ABB RAPID module: backup.MOD

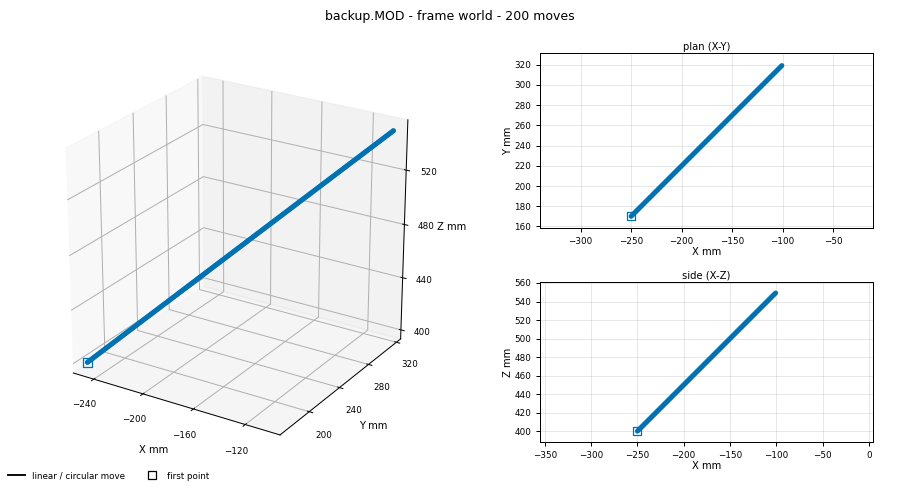
[picture p0: tool path of backup.MOD in frame world, 200 of 201 moves have a stored position in this frame; points joined in program order, loops and branches not executed]
MODULE MainModule
PERS tooldata Servo:=[TRUE,[[0,0,114.2],[1,0,0,0]],[0.215,[8.7,12.3,49.2],[1,0,0,0],0.00021,0.00024,0.00009]];
PERS tooldata tObject:=[TRUE,[[0,0,130],[0.707106781,-0.707106781,0,0]],[0.215,[8.7,12.3,49.2],[1,0,0,0],0.00021,0.00024,0.00009]];
PERS wobjdata handpos:= [FALSE,TRUE,"",[[-400,20,250],[1,0,0,0]],[[0,0,0],[1,0,0,0]]];


    PROC main()
        ConfL\Off;
        SingArea\Wrist;
        !Startpos
        MoveAbsJ [[95.3526,8.2285,12.3495,-7.77934,80.6461,5.41418],[87.0554,9E+09,9E+09,9E+09,9E+09,9E+09]] \NoEOffs, v1000, fine, wi_tGripper;
	    path;
    ENDPROC
    PROC path()

VAR robtarget t0 := [[150.0, 150.0, 150.0], [0, -1, 0, 0], [0,0,-1,4], [-96,9E+09,9E+09,9E+09,9E+09,9E+09]];
VAR robtarget t1 := [[150.75, 150.75, 150.75], [0, -1, 0, 0], [0,0,-1,4], [-96,9E+09,9E+09,9E+09,9E+09,9E+09]];
VAR robtarget t2 := [[151.5, 151.5, 151.5], [0, -1, 0, 0], [0,0,-1,4], [-96,9E+09,9E+09,9E+09,9E+09,9E+09]];
VAR robtarget t3 := [[152.25, 152.25, 152.25], [0, -1, 0, 0], [0,0,-1,4], [-96,9E+09,9E+09,9E+09,9E+09,9E+09]];
VAR robtarget t4 := [[153.0, 153.0, 153.0], [0, -1, 0, 0], [0,0,-1,4], [-96,9E+09,9E+09,9E+09,9E+09,9E+09]];
VAR robtarget t5 := [[153.75, 153.75, 153.75], [0, -1, 0, 0], [0,0,-1,4], [-96,9E+09,9E+09,9E+09,9E+09,9E+09]];
VAR robtarget t6 := [[154.5, 154.5, 154.5], [0, -1, 0, 0], [0,0,-1,4], [-96,9E+09,9E+09,9E+09,9E+09,9E+09]];
VAR robtarget t7 := [[155.25, 155.25, 155.25], [0, -1, 0, 0], [0,0,-1,4], [-96,9E+09,9E+09,9E+09,9E+09,9E+09]];
VAR robtarget t8 := [[156.0, 156.0, 156.0], [0, -1, 0, 0], [0,0,-1,4], [-96,9E+09,9E+09,9E+09,9E+09,9E+09]];
VAR robtarget t9 := [[156.75, 156.75, 156.75], [0, -1, 0, 0], [0,0,-1,4], [-96,9E+09,9E+09,9E+09,9E+09,9E+09]];
VAR robtarget t10 := [[157.5, 157.5, 157.5], [0, -1, 0, 0], [0,0,-1,4], [-96,9E+09,9E+09,9E+09,9E+09,9E+09]];
VAR robtarget t11 := [[158.25, 158.25, 158.25], [0, -1, 0, 0], [0,0,-1,4], [-96,9E+09,9E+09,9E+09,9E+09,9E+09]];
VAR robtarget t12 := [[159.0, 159.0, 159.0], [0, -1, 0, 0], [0,0,-1,4], [-96,9E+09,9E+09,9E+09,9E+09,9E+09]];
VAR robtarget t13 := [[159.75, 159.75, 159.75], [0, -1, 0, 0], [0,0,-1,4], [-96,9E+09,9E+09,9E+09,9E+09,9E+09]];
VAR robtarget t14 := [[160.5, 160.5, 160.5], [0, -1, 0, 0], [0,0,-1,4], [-96,9E+09,9E+09,9E+09,9E+09,9E+09]];
VAR robtarget t15 := [[161.25, 161.25, 161.25], [0, -1, 0, 0], [0,0,-1,4], [-96,9E+09,9E+09,9E+09,9E+09,9E+09]];
VAR robtarget t16 := [[162.0, 162.0, 162.0], [0, -1, 0, 0], [0,0,-1,4], [-96,9E+09,9E+09,9E+09,9E+09,9E+09]];
VAR robtarget t17 := [[162.75, 162.75, 162.75], [0, -1, 0, 0], [0,0,-1,4], [-96,9E+09,9E+09,9E+09,9E+09,9E+09]];a
VAR robtarget t18 := [[163.5, 163.5, 163.5], [0, -1, 0, 0], [0,0,-1,4], [-96,9E+09,9E+09,9E+09,9E+09,9E+09]];
VAR robtarget t19 := [[164.25, 164.25, 164.25], [0, -1, 0, 0], [0,0,-1,4], [-96,9E+09,9E+09,9E+09,9E+09,9E+09]];
VAR robtarget t20 := [[164.99999999999997, 164.99999999999997, 164.99999999999997], [0, -1, 0, 0], [0,0,-1,4], [-96,9E+09,9E+09,9E+09,9E+09,9E+09]];
VAR robtarget t21 := [[165.75, 165.75, 165.75], [0, -1, 0, 0], [0,0,-1,4], [-96,9E+09,9E+09,9E+09,9E+09,9E+09]];
VAR robtarget t22 := [[166.49999999999997, 166.49999999999997, 166.49999999999997], [0, -1, 0, 0], [0,0,-1,4], [-96,9E+09,9E+09,9E+09,9E+09,9E+09]];
VAR robtarget t23 := [[167.25, 167.25, 167.25], [0, -1, 0, 0], [0,0,-1,4], [-96,9E+09,9E+09,9E+09,9E+09,9E+09]];
VAR robtarget t24 := [[167.99999999999997, 167.99999999999997, 167.99999999999997], [0, -1, 0, 0], [0,0,-1,4], [-96,9E+09,9E+09,9E+09,9E+09,9E+09]];
VAR robtarget t25 := [[168.74999999999997, 168.74999999999997, 168.74999999999997], [0, -1, 0, 0], [0,0,-1,4], [-96,9E+09,9E+09,9E+09,9E+09,9E+09]];
VAR robtarget t26 := [[169.49999999999997, 169.49999999999997, 169.49999999999997], [0, -1, 0, 0], [0,0,-1,4], [-96,9E+09,9E+09,9E+09,9E+09,9E+09]];
VAR robtarget t27 := [[170.24999999999997, 170.24999999999997, 170.24999999999997], [0, -1, 0, 0], [0,0,-1,4], [-96,9E+09,9E+09,9E+09,9E+09,9E+09]];
VAR robtarget t28 := [[170.99999999999997, 170.99999999999997, 170.99999999999997], [0, -1, 0, 0], [0,0,-1,4], [-96,9E+09,9E+09,9E+09,9E+09,9E+09]];
VAR robtarget t29 := [[171.75, 171.75, 171.75], [0, -1, 0, 0], [0,0,-1,4], [-96,9E+09,9E+09,9E+09,9E+09,9E+09]];
VAR robtarget t30 := [[172.5, 172.5, 172.5], [0, -1, 0, 0], [0,0,-1,4], [-96,9E+09,9E+09,9E+09,9E+09,9E+09]];
VAR robtarget t31 := [[173.25, 173.25, 173.25], [0, -1, 0, 0], [0,0,-1,4], [-96,9E+09,9E+09,9E+09,9E+09,9E+09]];
VAR robtarget t32 := [[174.0, 174.0, 174.0], [0, -1, 0, 0], [0,0,-1,4], [-96,9E+09,9E+09,9E+09,9E+09,9E+09]];
VAR robtarget t33 := [[174.75, 174.75, 174.75], [0, -1, 0, 0], [0,0,-1,4], [-96,9E+09,9E+09,9E+09,9E+09,9E+09]];
VAR robtarget t34 := [[175.5, 175.5, 175.5], [0, -1, 0, 0], [0,0,-1,4], [-96,9E+09,9E+09,9E+09,9E+09,9E+09]];
VAR robtarget t35 := [[176.25, 176.25, 176.25], [0, -1, 0, 0], [0,0,-1,4], [-96,9E+09,9E+09,9E+09,9E+09,9E+09]];
VAR robtarget t36 := [[177.0, 177.0, 177.0], [0, -1, 0, 0], [0,0,-1,4], [-96,9E+09,9E+09,9E+09,9E+09,9E+09]];
VAR robtarget t37 := [[177.75, 177.75, 177.75], [0, -1, 0, 0], [0,0,-1,4], [-96,9E+09,9E+09,9E+09,9E+09,9E+09]];
VAR robtarget t38 := [[178.5, 178.5, 178.5], [0, -1, 0, 0], [0,0,-1,4], [-96,9E+09,9E+09,9E+09,9E+09,9E+09]];
VAR robtarget t39 := [[179.25, 179.25, 179.25], [0, -1, 0, 0], [0,0,-1,4], [-96,9E+09,9E+09,9E+09,9E+09,9E+09]];
VAR robtarget t40 := [[180.0, 180.0, 180.0], [0, -1, 0, 0], [0,0,-1,4], [-96,9E+09,9E+09,9E+09,9E+09,9E+09]];
VAR robtarget t41 := [[180.75, 180.75, 180.75], [0, -1, 0, 0], [0,0,-1,4], [-96,9E+09,9E+09,9E+09,9E+09,9E+09]];
VAR robtarget t42 := [[181.5, 181.5, 181.5], [0, -1, 0, 0], [0,0,-1,4], [-96,9E+09,9E+09,9E+09,9E+09,9E+09]];
VAR robtarget t43 := [[182.25, 182.25, 182.25], [0, -1, 0, 0], [0,0,-1,4], [-96,9E+09,9E+09,9E+09,9E+09,9E+09]];
VAR robtarget t44 := [[183.0, 183.0, 183.0], [0, -1, 0, 0], [0,0,-1,4], [-96,9E+09,9E+09,9E+09,9E+09,9E+09]];
VAR robtarget t45 := [[183.75, 183.75, 183.75], [0, -1, 0, 0], [0,0,-1,4], [-96,9E+09,9E+09,9E+09,9E+09,9E+09]];
VAR robtarget t46 := [[184.5, 184.5, 184.5], [0, -1, 0, 0], [0,0,-1,4], [-96,9E+09,9E+09,9E+09,9E+09,9E+09]];
VAR robtarget t47 := [[185.25, 185.25, 185.25], [0, -1, 0, 0], [0,0,-1,4], [-96,9E+09,9E+09,9E+09,9E+09,9E+09]];
VAR robtarget t48 := [[186.0, 186.0, 186.0], [0, -1, 0, 0], [0,0,-1,4], [-96,9E+09,9E+09,9E+09,9E+09,9E+09]];
VAR robtarget t49 := [[186.75, 186.75, 186.75], [0, -1, 0, 0], [0,0,-1,4], [-96,9E+09,9E+09,9E+09,9E+09,9E+09]];
VAR robtarget t50 := [[187.5, 187.5, 187.5], [0, -1, 0, 0], [0,0,-1,4], [-96,9E+09,9E+09,9E+09,9E+09,9E+09]];
VAR robtarget t51 := [[188.25, 188.25, 188.25], [0, -1, 0, 0], [0,0,-1,4], [-96,9E+09,9E+09,9E+09,9E+09,9E+09]];
VAR robtarget t52 := [[189.0, 189.0, 189.0], [0, -1, 0, 0], [0,0,-1,4], [-96,9E+09,9E+09,9E+09,9E+09,9E+09]];
VAR robtarget t53 := [[189.75, 189.75, 189.75], [0, -1, 0, 0], [0,0,-1,4], [-96,9E+09,9E+09,9E+09,9E+09,9E+09]];
VAR robtarget t54 := [[190.5, 190.5, 190.5], [0, -1, 0, 0], [0,0,-1,4], [-96,9E+09,9E+09,9E+09,9E+09,9E+09]];
VAR robtarget t55 := [[191.25, 191.25, 191.25], [0, -1, 0, 0], [0,0,-1,4], [-96,9E+09,9E+09,9E+09,9E+09,9E+09]];
VAR robtarget t56 := [[192.0, 192.0, 192.0], [0, -1, 0, 0], [0,0,-1,4], [-96,9E+09,9E+09,9E+09,9E+09,9E+09]];
VAR robtarget t57 := [[192.75, 192.75, 192.75], [0, -1, 0, 0], [0,0,-1,4], [-96,9E+09,9E+09,9E+09,9E+09,9E+09]];
VAR robtarget t58 := [[193.5, 193.5, 193.5], [0, -1, 0, 0], [0,0,-1,4], [-96,9E+09,9E+09,9E+09,9E+09,9E+09]];
VAR robtarget t59 := [[194.24999999999997, 194.24999999999997, 194.24999999999997], [0, -1, 0, 0], [0,0,-1,4], [-96,9E+09,9E+09,9E+09,9E+09,9E+09]];
VAR robtarget t60 := [[195.0, 195.0, 195.0], [0, -1, 0, 0], [0,0,-1,4], [-96,9E+09,9E+09,9E+09,9E+09,9E+09]];
VAR robtarget t61 := [[195.74999999999997, 195.74999999999997, 195.74999999999997], [0, -1, 0, 0], [0,0,-1,4], [-96,9E+09,9E+09,9E+09,9E+09,9E+09]];
VAR robtarget t62 := [[196.5, 196.5, 196.5], [0, -1, 0, 0], [0,0,-1,4], [-96,9E+09,9E+09,9E+09,9E+09,9E+09]];
VAR robtarget t63 := [[197.24999999999997, 197.24999999999997, 197.24999999999997], [0, -1, 0, 0], [0,0,-1,4], [-96,9E+09,9E+09,9E+09,9E+09,9E+09]];
VAR robtarget t64 := [[198.0, 198.0, 198.0], [0, -1, 0, 0], [0,0,-1,4], [-96,9E+09,9E+09,9E+09,9E+09,9E+09]];
VAR robtarget t65 := [[198.74999999999997, 198.74999999999997, 198.74999999999997], [0, -1, 0, 0], [0,0,-1,4], [-96,9E+09,9E+09,9E+09,9E+09,9E+09]];
VAR robtarget t66 := [[199.5, 199.5, 199.5], [0, -1, 0, 0], [0,0,-1,4], [-96,9E+09,9E+09,9E+09,9E+09,9E+09]];
VAR robtarget t67 := [[200.24999999999997, 200.24999999999997, 200.24999999999997], [0, -1, 0, 0], [0,0,-1,4], [-96,9E+09,9E+09,9E+09,9E+09,9E+09]];
VAR robtarget t68 := [[201.0, 201.0, 201.0], [0, -1, 0, 0], [0,0,-1,4], [-96,9E+09,9E+09,9E+09,9E+09,9E+09]];
VAR robtarget t69 := [[201.74999999999997, 201.74999999999997, 201.74999999999997], [0, -1, 0, 0], [0,0,-1,4], [-96,9E+09,9E+09,9E+09,9E+09,9E+09]];
VAR robtarget t70 := [[202.49999999999997, 202.49999999999997, 202.49999999999997], [0, -1, 0, 0], [0,0,-1,4], [-96,9E+09,9E+09,9E+09,9E+09,9E+09]];
VAR robtarget t71 := [[203.25, 203.25, 203.25], [0, -1, 0, 0], [0,0,-1,4], [-96,9E+09,9E+09,9E+09,9E+09,9E+09]];
VAR robtarget t72 := [[204.0, 204.0, 204.0], [0, -1, 0, 0], [0,0,-1,4], [-96,9E+09,9E+09,9E+09,9E+09,9E+09]];
VAR robtarget t73 := [[204.75, 204.75, 204.75], [0, -1, 0, 0], [0,0,-1,4], [-96,9E+09,9E+09,9E+09,9E+09,9E+09]];
VAR robtarget t74 := [[205.5, 205.5, 205.5], [0, -1, 0, 0], [0,0,-1,4], [-96,9E+09,9E+09,9E+09,9E+09,9E+09]];
VAR robtarget t75 := [[206.25, 206.25, 206.25], [0, -1, 0, 0], [0,0,-1,4], [-96,9E+09,9E+09,9E+09,9E+09,9E+09]];
VAR robtarget t76 := [[207.0, 207.0, 207.0], [0, -1, 0, 0], [0,0,-1,4], [-96,9E+09,9E+09,9E+09,9E+09,9E+09]];
VAR robtarget t77 := [[207.75, 207.75, 207.75], [0, -1, 0, 0], [0,0,-1,4], [-96,9E+09,9E+09,9E+09,9E+09,9E+09]];
VAR robtarget t78 := [[208.5, 208.5, 208.5], [0, -1, 0, 0], [0,0,-1,4], [-96,9E+09,9E+09,9E+09,9E+09,9E+09]];
VAR robtarget t79 := [[209.25, 209.25, 209.25], [0, -1, 0, 0], [0,0,-1,4], [-96,9E+09,9E+09,9E+09,9E+09,9E+09]];
VAR robtarget t80 := [[210.0, 210.0, 210.0], [0, -1, 0, 0], [0,0,-1,4], [-96,9E+09,9E+09,9E+09,9E+09,9E+09]];
VAR robtarget t81 := [[210.75, 210.75, 210.75], [0, -1, 0, 0], [0,0,-1,4], [-96,9E+09,9E+09,9E+09,9E+09,9E+09]];
VAR robtarget t82 := [[211.5, 211.5, 211.5], [0, -1, 0, 0], [0,0,-1,4], [-96,9E+09,9E+09,9E+09,9E+09,9E+09]];
VAR robtarget t83 := [[212.25, 212.25, 212.25], [0, -1, 0, 0], [0,0,-1,4], [-96,9E+09,9E+09,9E+09,9E+09,9E+09]];
VAR robtarget t84 := [[213.0, 213.0, 213.0], [0, -1, 0, 0], [0,0,-1,4], [-96,9E+09,9E+09,9E+09,9E+09,9E+09]];
VAR robtarget t85 := [[213.75, 213.75, 213.75], [0, -1, 0, 0], [0,0,-1,4], [-96,9E+09,9E+09,9E+09,9E+09,9E+09]];
VAR robtarget t86 := [[214.5, 214.5, 214.5], [0, -1, 0, 0], [0,0,-1,4], [-96,9E+09,9E+09,9E+09,9E+09,9E+09]];
VAR robtarget t87 := [[215.25, 215.25, 215.25], [0, -1, 0, 0], [0,0,-1,4], [-96,9E+09,9E+09,9E+09,9E+09,9E+09]];
VAR robtarget t88 := [[216.0, 216.0, 216.0], [0, -1, 0, 0], [0,0,-1,4], [-96,9E+09,9E+09,9E+09,9E+09,9E+09]];
VAR robtarget t89 := [[216.75, 216.75, 216.75], [0, -1, 0, 0], [0,0,-1,4], [-96,9E+09,9E+09,9E+09,9E+09,9E+09]];
VAR robtarget t90 := [[217.5, 217.5, 217.5], [0, -1, 0, 0], [0,0,-1,4], [-96,9E+09,9E+09,9E+09,9E+09,9E+09]];
VAR robtarget t91 := [[218.25, 218.25, 218.25], [0, -1, 0, 0], [0,0,-1,4], [-96,9E+09,9E+09,9E+09,9E+09,9E+09]];
VAR robtarget t92 := [[219.0, 219.0, 219.0], [0, -1, 0, 0], [0,0,-1,4], [-96,9E+09,9E+09,9E+09,9E+09,9E+09]];
VAR robtarget t93 := [[219.75, 219.75, 219.75], [0, -1, 0, 0], [0,0,-1,4], [-96,9E+09,9E+09,9E+09,9E+09,9E+09]];
VAR robtarget t94 := [[220.5, 220.5, 220.5], [0, -1, 0, 0], [0,0,-1,4], [-96,9E+09,9E+09,9E+09,9E+09,9E+09]];
VAR robtarget t95 := [[221.25, 221.25, 221.25], [0, -1, 0, 0], [0,0,-1,4], [-96,9E+09,9E+09,9E+09,9E+09,9E+09]];
VAR robtarget t96 := [[222.0, 222.0, 222.0], [0, -1, 0, 0], [0,0,-1,4], [-96,9E+09,9E+09,9E+09,9E+09,9E+09]];
VAR robtarget t97 := [[222.75, 222.75, 222.75], [0, -1, 0, 0], [0,0,-1,4], [-96,9E+09,9E+09,9E+09,9E+09,9E+09]];
VAR robtarget t98 := [[223.49999999999997, 223.49999999999997, 223.49999999999997], [0, -1, 0, 0], [0,0,-1,4], [-96,9E+09,9E+09,9E+09,9E+09,9E+09]];
VAR robtarget t99 := [[224.25, 224.25, 224.25], [0, -1, 0, 0], [0,0,-1,4], [-96,9E+09,9E+09,9E+09,9E+09,9E+09]];
VAR robtarget t100 := [[224.99999999999997, 224.99999999999997, 224.99999999999997], [0, -1, 0, 0], [0,0,-1,4], [-96,9E+09,9E+09,9E+09,9E+09,9E+09]];
VAR robtarget t101 := [[225.75, 225.75, 225.75], [0, -1, 0, 0], [0,0,-1,4], [-96,9E+09,9E+09,9E+09,9E+09,9E+09]];
VAR robtarget t102 := [[226.49999999999997, 226.49999999999997, 226.49999999999997], [0, -1, 0, 0], [0,0,-1,4], [-96,9E+09,9E+09,9E+09,9E+09,9E+09]];
VAR robtarget t103 := [[227.25, 227.25, 227.25], [0, -1, 0, 0], [0,0,-1,4], [-96,9E+09,9E+09,9E+09,9E+09,9E+09]];
VAR robtarget t104 := [[227.99999999999997, 227.99999999999997, 227.99999999999997], [0, -1, 0, 0], [0,0,-1,4], [-96,9E+09,9E+09,9E+09,9E+09,9E+09]];
VAR robtarget t105 := [[228.75, 228.75, 228.75], [0, -1, 0, 0], [0,0,-1,4], [-96,9E+09,9E+09,9E+09,9E+09,9E+09]];
VAR robtarget t106 := [[229.49999999999997, 229.49999999999997, 229.49999999999997], [0, -1, 0, 0], [0,0,-1,4], [-96,9E+09,9E+09,9E+09,9E+09,9E+09]];
VAR robtarget t107 := [[230.25, 230.25, 230.25], [0, -1, 0, 0], [0,0,-1,4], [-96,9E+09,9E+09,9E+09,9E+09,9E+09]];
VAR robtarget t108 := [[230.99999999999997, 230.99999999999997, 230.99999999999997], [0, -1, 0, 0], [0,0,-1,4], [-96,9E+09,9E+09,9E+09,9E+09,9E+09]];
VAR robtarget t109 := [[231.75, 231.75, 231.75], [0, -1, 0, 0], [0,0,-1,4], [-96,9E+09,9E+09,9E+09,9E+09,9E+09]];
VAR robtarget t110 := [[232.49999999999997, 232.49999999999997, 232.49999999999997], [0, -1, 0, 0], [0,0,-1,4], [-96,9E+09,9E+09,9E+09,9E+09,9E+09]];
VAR robtarget t111 := [[233.25, 233.25, 233.25], [0, -1, 0, 0], [0,0,-1,4], [-96,9E+09,9E+09,9E+09,9E+09,9E+09]];
VAR robtarget t112 := [[234.0, 234.0, 234.0], [0, -1, 0, 0], [0,0,-1,4], [-96,9E+09,9E+09,9E+09,9E+09,9E+09]];
VAR robtarget t113 := [[234.75, 234.75, 234.75], [0, -1, 0, 0], [0,0,-1,4], [-96,9E+09,9E+09,9E+09,9E+09,9E+09]];
VAR robtarget t114 := [[235.5, 235.5, 235.5], [0, -1, 0, 0], [0,0,-1,4], [-96,9E+09,9E+09,9E+09,9E+09,9E+09]];
VAR robtarget t115 := [[236.25000000000003, 236.25000000000003, 236.25000000000003], [0, -1, 0, 0], [0,0,-1,4], [-96,9E+09,9E+09,9E+09,9E+09,9E+09]];
VAR robtarget t116 := [[237.0, 237.0, 237.0], [0, -1, 0, 0], [0,0,-1,4], [-96,9E+09,9E+09,9E+09,9E+09,9E+09]];
VAR robtarget t117 := [[237.75000000000003, 237.75000000000003, 237.75000000000003], [0, -1, 0, 0], [0,0,-1,4], [-96,9E+09,9E+09,9E+09,9E+09,9E+09]];
VAR robtarget t118 := [[238.5, 238.5, 238.5], [0, -1, 0, 0], [0,0,-1,4], [-96,9E+09,9E+09,9E+09,9E+09,9E+09]];
VAR robtarget t119 := [[239.25, 239.25, 239.25], [0, -1, 0, 0], [0,0,-1,4], [-96,9E+09,9E+09,9E+09,9E+09,9E+09]];
VAR robtarget t120 := [[240.0, 240.0, 240.0], [0, -1, 0, 0], [0,0,-1,4], [-96,9E+09,9E+09,9E+09,9E+09,9E+09]];
VAR robtarget t121 := [[240.75, 240.75, 240.75], [0, -1, 0, 0], [0,0,-1,4], [-96,9E+09,9E+09,9E+09,9E+09,9E+09]];
VAR robtarget t122 := [[241.5, 241.5, 241.5], [0, -1, 0, 0], [0,0,-1,4], [-96,9E+09,9E+09,9E+09,9E+09,9E+09]];
VAR robtarget t123 := [[242.25, 242.25, 242.25], [0, -1, 0, 0], [0,0,-1,4], [-96,9E+09,9E+09,9E+09,9E+09,9E+09]];
VAR robtarget t124 := [[243.0, 243.0, 243.0], [0, -1, 0, 0], [0,0,-1,4], [-96,9E+09,9E+09,9E+09,9E+09,9E+09]];
VAR robtarget t125 := [[243.75, 243.75, 243.75], [0, -1, 0, 0], [0,0,-1,4], [-96,9E+09,9E+09,9E+09,9E+09,9E+09]];
VAR robtarget t126 := [[244.5, 244.5, 244.5], [0, -1, 0, 0], [0,0,-1,4], [-96,9E+09,9E+09,9E+09,9E+09,9E+09]];
VAR robtarget t127 := [[245.25, 245.25, 245.25], [0, -1, 0, 0], [0,0,-1,4], [-96,9E+09,9E+09,9E+09,9E+09,9E+09]];
VAR robtarget t128 := [[246.0, 246.0, 246.0], [0, -1, 0, 0], [0,0,-1,4], [-96,9E+09,9E+09,9E+09,9E+09,9E+09]];
VAR robtarget t129 := [[246.75, 246.75, 246.75], [0, -1, 0, 0], [0,0,-1,4], [-96,9E+09,9E+09,9E+09,9E+09,9E+09]];
VAR robtarget t130 := [[247.5, 247.5, 247.5], [0, -1, 0, 0], [0,0,-1,4], [-96,9E+09,9E+09,9E+09,9E+09,9E+09]];
VAR robtarget t131 := [[248.25, 248.25, 248.25], [0, -1, 0, 0], [0,0,-1,4], [-96,9E+09,9E+09,9E+09,9E+09,9E+09]];
VAR robtarget t132 := [[249.0, 249.0, 249.0], [0, -1, 0, 0], [0,0,-1,4], [-96,9E+09,9E+09,9E+09,9E+09,9E+09]];
VAR robtarget t133 := [[249.75, 249.75, 249.75], [0, -1, 0, 0], [0,0,-1,4], [-96,9E+09,9E+09,9E+09,9E+09,9E+09]];
VAR robtarget t134 := [[250.5, 250.5, 250.5], [0, -1, 0, 0], [0,0,-1,4], [-96,9E+09,9E+09,9E+09,9E+09,9E+09]];
VAR robtarget t135 := [[251.24999999999997, 251.24999999999997, 251.24999999999997], [0, -1, 0, 0], [0,0,-1,4], [-96,9E+09,9E+09,9E+09,9E+09,9E+09]];
VAR robtarget t136 := [[252.0, 252.0, 252.0], [0, -1, 0, 0], [0,0,-1,4], [-96,9E+09,9E+09,9E+09,9E+09,9E+09]];
VAR robtarget t137 := [[252.75000000000003, 252.75000000000003, 252.75000000000003], [0, -1, 0, 0], [0,0,-1,4], [-96,9E+09,9E+09,9E+09,9E+09,9E+09]];
VAR robtarget t138 := [[253.5, 253.5, 253.5], [0, -1, 0, 0], [0,0,-1,4], [-96,9E+09,9E+09,9E+09,9E+09,9E+09]];
VAR robtarget t139 := [[254.24999999999997, 254.24999999999997, 254.24999999999997], [0, -1, 0, 0], [0,0,-1,4], [-96,9E+09,9E+09,9E+09,9E+09,9E+09]];
VAR robtarget t140 := [[255.0, 255.0, 255.0], [0, -1, 0, 0], [0,0,-1,4], [-96,9E+09,9E+09,9E+09,9E+09,9E+09]];
VAR robtarget t141 := [[255.74999999999997, 255.74999999999997, 255.74999999999997], [0, -1, 0, 0], [0,0,-1,4], [-96,9E+09,9E+09,9E+09,9E+09,9E+09]];
VAR robtarget t142 := [[256.5, 256.5, 256.5], [0, -1, 0, 0], [0,0,-1,4], [-96,9E+09,9E+09,9E+09,9E+09,9E+09]];
VAR robtarget t143 := [[257.25, 257.25, 257.25], [0, -1, 0, 0], [0,0,-1,4], [-96,9E+09,9E+09,9E+09,9E+09,9E+09]];
VAR robtarget t144 := [[258.0, 258.0, 258.0], [0, -1, 0, 0], [0,0,-1,4], [-96,9E+09,9E+09,9E+09,9E+09,9E+09]];
VAR robtarget t145 := [[258.75, 258.75, 258.75], [0, -1, 0, 0], [0,0,-1,4], [-96,9E+09,9E+09,9E+09,9E+09,9E+09]];
VAR robtarget t146 := [[259.5, 259.5, 259.5], [0, -1, 0, 0], [0,0,-1,4], [-96,9E+09,9E+09,9E+09,9E+09,9E+09]];
VAR robtarget t147 := [[260.25, 260.25, 260.25], [0, -1, 0, 0], [0,0,-1,4], [-96,9E+09,9E+09,9E+09,9E+09,9E+09]];
VAR robtarget t148 := [[261.0, 261.0, 261.0], [0, -1, 0, 0], [0,0,-1,4], [-96,9E+09,9E+09,9E+09,9E+09,9E+09]];
VAR robtarget t149 := [[261.75, 261.75, 261.75], [0, -1, 0, 0], [0,0,-1,4], [-96,9E+09,9E+09,9E+09,9E+09,9E+09]];
VAR robtarget t150 := [[262.5, 262.5, 262.5], [0, -1, 0, 0], [0,0,-1,4], [-96,9E+09,9E+09,9E+09,9E+09,9E+09]];
VAR robtarget t151 := [[263.25, 263.25, 263.25], [0, -1, 0, 0], [0,0,-1,4], [-96,9E+09,9E+09,9E+09,9E+09,9E+09]];
VAR robtarget t152 := [[264.0, 264.0, 264.0], [0, -1, 0, 0], [0,0,-1,4], [-96,9E+09,9E+09,9E+09,9E+09,9E+09]];
VAR robtarget t153 := [[264.75, 264.75, 264.75], [0, -1, 0, 0], [0,0,-1,4], [-96,9E+09,9E+09,9E+09,9E+09,9E+09]];
VAR robtarget t154 := [[265.5, 265.5, 265.5], [0, -1, 0, 0], [0,0,-1,4], [-96,9E+09,9E+09,9E+09,9E+09,9E+09]];
VAR robtarget t155 := [[266.25, 266.25, 266.25], [0, -1, 0, 0], [0,0,-1,4], [-96,9E+09,9E+09,9E+09,9E+09,9E+09]];
VAR robtarget t156 := [[267.0, 267.0, 267.0], [0, -1, 0, 0], [0,0,-1,4], [-96,9E+09,9E+09,9E+09,9E+09,9E+09]];
VAR robtarget t157 := [[267.75, 267.75, 267.75], [0, -1, 0, 0], [0,0,-1,4], [-96,9E+09,9E+09,9E+09,9E+09,9E+09]];
VAR robtarget t158 := [[268.5, 268.5, 268.5], [0, -1, 0, 0], [0,0,-1,4], [-96,9E+09,9E+09,9E+09,9E+09,9E+09]];
VAR robtarget t159 := [[269.25, 269.25, 269.25], [0, -1, 0, 0], [0,0,-1,4], [-96,9E+09,9E+09,9E+09,9E+09,9E+09]];
VAR robtarget t160 := [[270.0, 270.0, 270.0], [0, -1, 0, 0], [0,0,-1,4], [-96,9E+09,9E+09,9E+09,9E+09,9E+09]];
VAR robtarget t161 := [[270.75, 270.75, 270.75], [0, -1, 0, 0], [0,0,-1,4], [-96,9E+09,9E+09,9E+09,9E+09,9E+09]];
VAR robtarget t162 := [[271.49999999999994, 271.49999999999994, 271.49999999999994], [0, -1, 0, 0], [0,0,-1,4], [-96,9E+09,9E+09,9E+09,9E+09,9E+09]];
VAR robtarget t163 := [[272.25, 272.25, 272.25], [0, -1, 0, 0], [0,0,-1,4], [-96,9E+09,9E+09,9E+09,9E+09,9E+09]];
VAR robtarget t164 := [[273.0, 273.0, 273.0], [0, -1, 0, 0], [0,0,-1,4], [-96,9E+09,9E+09,9E+09,9E+09,9E+09]];
VAR robtarget t165 := [[273.75, 273.75, 273.75], [0, -1, 0, 0], [0,0,-1,4], [-96,9E+09,9E+09,9E+09,9E+09,9E+09]];
VAR robtarget t166 := [[274.49999999999994, 274.49999999999994, 274.49999999999994], [0, -1, 0, 0], [0,0,-1,4], [-96,9E+09,9E+09,9E+09,9E+09,9E+09]];
VAR robtarget t167 := [[275.25, 275.25, 275.25], [0, -1, 0, 0], [0,0,-1,4], [-96,9E+09,9E+09,9E+09,9E+09,9E+09]];
VAR robtarget t168 := [[276.0, 276.0, 276.0], [0, -1, 0, 0], [0,0,-1,4], [-96,9E+09,9E+09,9E+09,9E+09,9E+09]];
VAR robtarget t169 := [[276.75, 276.75, 276.75], [0, -1, 0, 0], [0,0,-1,4], [-96,9E+09,9E+09,9E+09,9E+09,9E+09]];
VAR robtarget t170 := [[277.49999999999994, 277.49999999999994, 277.49999999999994], [0, -1, 0, 0], [0,0,-1,4], [-96,9E+09,9E+09,9E+09,9E+09,9E+09]];
VAR robtarget t171 := [[278.25, 278.25, 278.25], [0, -1, 0, 0], [0,0,-1,4], [-96,9E+09,9E+09,9E+09,9E+09,9E+09]];
VAR robtarget t172 := [[279.0, 279.0, 279.0], [0, -1, 0, 0], [0,0,-1,4], [-96,9E+09,9E+09,9E+09,9E+09,9E+09]];
VAR robtarget t173 := [[279.75, 279.75, 279.75], [0, -1, 0, 0], [0,0,-1,4], [-96,9E+09,9E+09,9E+09,9E+09,9E+09]];
VAR robtarget t174 := [[280.5, 280.5, 280.5], [0, -1, 0, 0], [0,0,-1,4], [-96,9E+09,9E+09,9E+09,9E+09,9E+09]];
VAR robtarget t175 := [[281.25, 281.25, 281.25], [0, -1, 0, 0], [0,0,-1,4], [-96,9E+09,9E+09,9E+09,9E+09,9E+09]];
VAR robtarget t176 := [[282.0, 282.0, 282.0], [0, -1, 0, 0], [0,0,-1,4], [-96,9E+09,9E+09,9E+09,9E+09,9E+09]];
VAR robtarget t177 := [[282.75, 282.75, 282.75], [0, -1, 0, 0], [0,0,-1,4], [-96,9E+09,9E+09,9E+09,9E+09,9E+09]];
VAR robtarget t178 := [[283.5, 283.5, 283.5], [0, -1, 0, 0], [0,0,-1,4], [-96,9E+09,9E+09,9E+09,9E+09,9E+09]];
VAR robtarget t179 := [[284.25, 284.25, 284.25], [0, -1, 0, 0], [0,0,-1,4], [-96,9E+09,9E+09,9E+09,9E+09,9E+09]];
VAR robtarget t180 := [[285.00000000000006, 285.00000000000006, 285.00000000000006], [0, -1, 0, 0], [0,0,-1,4], [-96,9E+09,9E+09,9E+09,9E+09,9E+09]];
VAR robtarget t181 := [[285.75, 285.75, 285.75], [0, -1, 0, 0], [0,0,-1,4], [-96,9E+09,9E+09,9E+09,9E+09,9E+09]];
VAR robtarget t182 := [[286.5, 286.5, 286.5], [0, -1, 0, 0], [0,0,-1,4], [-96,9E+09,9E+09,9E+09,9E+09,9E+09]];
VAR robtarget t183 := [[287.25, 287.25, 287.25], [0, -1, 0, 0], [0,0,-1,4], [-96,9E+09,9E+09,9E+09,9E+09,9E+09]];
VAR robtarget t184 := [[288.00000000000006, 288.00000000000006, 288.00000000000006], [0, -1, 0, 0], [0,0,-1,4], [-96,9E+09,9E+09,9E+09,9E+09,9E+09]];
VAR robtarget t185 := [[288.75, 288.75, 288.75], [0, -1, 0, 0], [0,0,-1,4], [-96,9E+09,9E+09,9E+09,9E+09,9E+09]];
VAR robtarget t186 := [[289.5, 289.5, 289.5], [0, -1, 0, 0], [0,0,-1,4], [-96,9E+09,9E+09,9E+09,9E+09,9E+09]];
VAR robtarget t187 := [[290.25, 290.25, 290.25], [0, -1, 0, 0], [0,0,-1,4], [-96,9E+09,9E+09,9E+09,9E+09,9E+09]];
VAR robtarget t188 := [[291.00000000000006, 291.00000000000006, 291.00000000000006], [0, -1, 0, 0], [0,0,-1,4], [-96,9E+09,9E+09,9E+09,9E+09,9E+09]];
VAR robtarget t189 := [[291.75, 291.75, 291.75], [0, -1, 0, 0], [0,0,-1,4], [-96,9E+09,9E+09,9E+09,9E+09,9E+09]];
VAR robtarget t190 := [[292.5, 292.5, 292.5], [0, -1, 0, 0], [0,0,-1,4], [-96,9E+09,9E+09,9E+09,9E+09,9E+09]];
VAR robtarget t191 := [[293.25, 293.25, 293.25], [0, -1, 0, 0], [0,0,-1,4], [-96,9E+09,9E+09,9E+09,9E+09,9E+09]];
VAR robtarget t192 := [[294.00000000000006, 294.00000000000006, 294.00000000000006], [0, -1, 0, 0], [0,0,-1,4], [-96,9E+09,9E+09,9E+09,9E+09,9E+09]];
VAR robtarget t193 := [[294.74999999999994, 294.74999999999994, 294.74999999999994], [0, -1, 0, 0], [0,0,-1,4], [-96,9E+09,9E+09,9E+09,9E+09,9E+09]];
VAR robtarget t194 := [[295.5, 295.5, 295.5], [0, -1, 0, 0], [0,0,-1,4], [-96,9E+09,9E+09,9E+09,9E+09,9E+09]];
VAR robtarget t195 := [[296.25, 296.25, 296.25], [0, -1, 0, 0], [0,0,-1,4], [-96,9E+09,9E+09,9E+09,9E+09,9E+09]];
VAR robtarget t196 := [[297.0, 297.0, 297.0], [0, -1, 0, 0], [0,0,-1,4], [-96,9E+09,9E+09,9E+09,9E+09,9E+09]];
VAR robtarget t197 := [[297.74999999999994, 297.74999999999994, 297.74999999999994], [0, -1, 0, 0], [0,0,-1,4], [-96,9E+09,9E+09,9E+09,9E+09,9E+09]];
VAR robtarget t198 := [[298.5, 298.5, 298.5], [0, -1, 0, 0], [0,0,-1,4], [-96,9E+09,9E+09,9E+09,9E+09,9E+09]];
VAR robtarget t199 := [[299.25, 299.25, 299.25], [0, -1, 0, 0], [0,0,-1,4], [-96,9E+09,9E+09,9E+09,9E+09,9E+09]];MoveL t0, v100\V:=100.000, z1, wi_tGripper, \WObj:=handpos;
MoveL t1, v100\V:=100.000, z1, wi_tGripper, \WObj:=handpos;
MoveL t2, v100\V:=100.000, z1, wi_tGripper, \WObj:=handpos;
MoveL t3, v100\V:=100.000, z1, wi_tGripper, \WObj:=handpos;
MoveL t4, v100\V:=100.000, z1, wi_tGripper, \WObj:=handpos;
MoveL t5, v100\V:=100.000, z1, wi_tGripper, \WObj:=handpos;
MoveL t6, v100\V:=100.000, z1, wi_tGripper, \WObj:=handpos;
MoveL t7, v100\V:=100.000, z1, wi_tGripper, \WObj:=handpos;
MoveL t8, v100\V:=100.000, z1, wi_tGripper, \WObj:=handpos;
MoveL t9, v100\V:=100.000, z1, wi_tGripper, \WObj:=handpos;
MoveL t10, v100\V:=100.000, z1, wi_tGripper, \WObj:=handpos;
MoveL t11, v100\V:=100.000, z1, wi_tGripper, \WObj:=handpos;
MoveL t12, v100\V:=100.000, z1, wi_tGripper, \WObj:=handpos;
MoveL t13, v100\V:=100.000, z1, wi_tGripper, \WObj:=handpos;
MoveL t14, v100\V:=100.000, z1, wi_tGripper, \WObj:=handpos;
MoveL t15, v100\V:=100.000, z1, wi_tGripper, \WObj:=handpos;
MoveL t16, v100\V:=100.000, z1, wi_tGripper, \WObj:=handpos;
MoveL t17, v100\V:=100.000, z1, wi_tGripper, \WObj:=handpos;
MoveL t18, v100\V:=100.000, z1, wi_tGripper, \WObj:=handpos;
MoveL t19, v100\V:=100.000, z1, wi_tGripper, \WObj:=handpos;
MoveL t20, v100\V:=100.000, z1, wi_tGripper, \WObj:=handpos;
MoveL t21, v100\V:=100.000, z1, wi_tGripper, \WObj:=handpos;
MoveL t22, v100\V:=100.000, z1, wi_tGripper, \WObj:=handpos;
MoveL t23, v100\V:=100.000, z1, wi_tGripper, \WObj:=handpos;
MoveL t24, v100\V:=100.000, z1, wi_tGripper, \WObj:=handpos;
MoveL t25, v100\V:=100.000, z1, wi_tGripper, \WObj:=handpos;
MoveL t26, v100\V:=100.000, z1, wi_tGripper, \WObj:=handpos;
MoveL t27, v100\V:=100.000, z1, wi_tGripper, \WObj:=handpos;
MoveL t28, v100\V:=100.000, z1, wi_tGripper, \WObj:=handpos;
MoveL t29, v100\V:=100.000, z1, wi_tGripper, \WObj:=handpos;
MoveL t30, v100\V:=100.000, z1, wi_tGripper, \WObj:=handpos;
MoveL t31, v100\V:=100.000, z1, wi_tGripper, \WObj:=handpos;
MoveL t32, v100\V:=100.000, z1, wi_tGripper, \WObj:=handpos;
MoveL t33, v100\V:=100.000, z1, wi_tGripper, \WObj:=handpos;
MoveL t34, v100\V:=100.000, z1, wi_tGripper, \WObj:=handpos;
MoveL t35, v100\V:=100.000, z1, wi_tGripper, \WObj:=handpos;
MoveL t36, v100\V:=100.000, z1, wi_tGripper, \WObj:=handpos;
MoveL t37, v100\V:=100.000, z1, wi_tGripper, \WObj:=handpos;
MoveL t38, v100\V:=100.000, z1, wi_tGripper, \WObj:=handpos;
MoveL t39, v100\V:=100.000, z1, wi_tGripper, \WObj:=handpos;
MoveL t40, v100\V:=100.000, z1, wi_tGripper, \WObj:=handpos;
MoveL t41, v100\V:=100.000, z1, wi_tGripper, \WObj:=handpos;
MoveL t42, v100\V:=100.000, z1, wi_tGripper, \WObj:=handpos;
MoveL t43, v100\V:=100.000, z1, wi_tGripper, \WObj:=handpos;
MoveL t44, v100\V:=100.000, z1, wi_tGripper, \WObj:=handpos;
MoveL t45, v100\V:=100.000, z1, wi_tGripper, \WObj:=handpos;
MoveL t46, v100\V:=100.000, z1, wi_tGripper, \WObj:=handpos;
MoveL t47, v100\V:=100.000, z1, wi_tGripper, \WObj:=handpos;
MoveL t48, v100\V:=100.000, z1, wi_tGripper, \WObj:=handpos;
MoveL t49, v100\V:=100.000, z1, wi_tGripper, \WObj:=handpos;
MoveL t50, v100\V:=100.000, z1, wi_tGripper, \WObj:=handpos;
MoveL t51, v100\V:=100.000, z1, wi_tGripper, \WObj:=handpos;
MoveL t52, v100\V:=100.000, z1, wi_tGripper, \WObj:=handpos;
MoveL t53, v100\V:=100.000, z1, wi_tGripper, \WObj:=handpos;
MoveL t54, v100\V:=100.000, z1, wi_tGripper, \WObj:=handpos;
MoveL t55, v100\V:=100.000, z1, wi_tGripper, \WObj:=handpos;
MoveL t56, v100\V:=100.000, z1, wi_tGripper, \WObj:=handpos;
MoveL t57, v100\V:=100.000, z1, wi_tGripper, \WObj:=handpos;
MoveL t58, v100\V:=100.000, z1, wi_tGripper, \WObj:=handpos;
MoveL t59, v100\V:=100.000, z1, wi_tGripper, \WObj:=handpos;
MoveL t60, v100\V:=100.000, z1, wi_tGripper, \WObj:=handpos;
MoveL t61, v100\V:=100.000, z1, wi_tGripper, \WObj:=handpos;
MoveL t62, v100\V:=100.000, z1, wi_tGripper, \WObj:=handpos;
MoveL t63, v100\V:=100.000, z1, wi_tGripper, \WObj:=handpos;
MoveL t64, v100\V:=100.000, z1, wi_tGripper, \WObj:=handpos;
MoveL t65, v100\V:=100.000, z1, wi_tGripper, \WObj:=handpos;
MoveL t66, v100\V:=100.000, z1, wi_tGripper, \WObj:=handpos;
MoveL t67, v100\V:=100.000, z1, wi_tGripper, \WObj:=handpos;
MoveL t68, v100\V:=100.000, z1, wi_tGripper, \WObj:=handpos;
MoveL t69, v100\V:=100.000, z1, wi_tGripper, \WObj:=handpos;
MoveL t70, v100\V:=100.000, z1, wi_tGripper, \WObj:=handpos;
MoveL t71, v100\V:=100.000, z1, wi_tGripper, \WObj:=handpos;
MoveL t72, v100\V:=100.000, z1, wi_tGripper, \WObj:=handpos;
MoveL t73, v100\V:=100.000, z1, wi_tGripper, \WObj:=handpos;
MoveL t74, v100\V:=100.000, z1, wi_tGripper, \WObj:=handpos;
MoveL t75, v100\V:=100.000, z1, wi_tGripper, \WObj:=handpos;
MoveL t76, v100\V:=100.000, z1, wi_tGripper, \WObj:=handpos;
MoveL t77, v100\V:=100.000, z1, wi_tGripper, \WObj:=handpos;
MoveL t78, v100\V:=100.000, z1, wi_tGripper, \WObj:=handpos;
MoveL t79, v100\V:=100.000, z1, wi_tGripper, \WObj:=handpos;
MoveL t80, v100\V:=100.000, z1, wi_tGripper, \WObj:=handpos;
MoveL t81, v100\V:=100.000, z1, wi_tGripper, \WObj:=handpos;
MoveL t82, v100\V:=100.000, z1, wi_tGripper, \WObj:=handpos;
MoveL t83, v100\V:=100.000, z1, wi_tGripper, \WObj:=handpos;
MoveL t84, v100\V:=100.000, z1, wi_tGripper, \WObj:=handpos;
MoveL t85, v100\V:=100.000, z1, wi_tGripper, \WObj:=handpos;
MoveL t86, v100\V:=100.000, z1, wi_tGripper, \WObj:=handpos;
MoveL t87, v100\V:=100.000, z1, wi_tGripper, \WObj:=handpos;
MoveL t88, v100\V:=100.000, z1, wi_tGripper, \WObj:=handpos;
MoveL t89, v100\V:=100.000, z1, wi_tGripper, \WObj:=handpos;
MoveL t90, v100\V:=100.000, z1, wi_tGripper, \WObj:=handpos;
MoveL t91, v100\V:=100.000, z1, wi_tGripper, \WObj:=handpos;
MoveL t92, v100\V:=100.000, z1, wi_tGripper, \WObj:=handpos;
MoveL t93, v100\V:=100.000, z1, wi_tGripper, \WObj:=handpos;
MoveL t94, v100\V:=100.000, z1, wi_tGripper, \WObj:=handpos;
MoveL t95, v100\V:=100.000, z1, wi_tGripper, \WObj:=handpos;
MoveL t96, v100\V:=100.000, z1, wi_tGripper, \WObj:=handpos;
MoveL t97, v100\V:=100.000, z1, wi_tGripper, \WObj:=handpos;
MoveL t98, v100\V:=100.000, z1, wi_tGripper, \WObj:=handpos;
MoveL t99, v100\V:=100.000, z1, wi_tGripper, \WObj:=handpos;
MoveL t100, v100\V:=100.000, z1, wi_tGripper, \WObj:=handpos;
MoveL t101, v100\V:=100.000, z1, wi_tGripper, \WObj:=handpos;
MoveL t102, v100\V:=100.000, z1, wi_tGripper, \WObj:=handpos;
MoveL t103, v100\V:=100.000, z1, wi_tGripper, \WObj:=handpos;
MoveL t104, v100\V:=100.000, z1, wi_tGripper, \WObj:=handpos;
MoveL t105, v100\V:=100.000, z1, wi_tGripper, \WObj:=handpos;
MoveL t106, v100\V:=100.000, z1, wi_tGripper, \WObj:=handpos;
MoveL t107, v100\V:=100.000, z1, wi_tGripper, \WObj:=handpos;
MoveL t108, v100\V:=100.000, z1, wi_tGripper, \WObj:=handpos;
MoveL t109, v100\V:=100.000, z1, wi_tGripper, \WObj:=handpos;
MoveL t110, v100\V:=100.000, z1, wi_tGripper, \WObj:=handpos;
MoveL t111, v100\V:=100.000, z1, wi_tGripper, \WObj:=handpos;
MoveL t112, v100\V:=100.000, z1, wi_tGripper, \WObj:=handpos;
MoveL t113, v100\V:=100.000, z1, wi_tGripper, \WObj:=handpos;
MoveL t114, v100\V:=100.000, z1, wi_tGripper, \WObj:=handpos;
MoveL t115, v100\V:=100.000, z1, wi_tGripper, \WObj:=handpos;
MoveL t116, v100\V:=100.000, z1, wi_tGripper, \WObj:=handpos;
MoveL t117, v100\V:=100.000, z1, wi_tGripper, \WObj:=handpos;
MoveL t118, v100\V:=100.000, z1, wi_tGripper, \WObj:=handpos;
MoveL t119, v100\V:=100.000, z1, wi_tGripper, \WObj:=handpos;
MoveL t120, v100\V:=100.000, z1, wi_tGripper, \WObj:=handpos;
MoveL t121, v100\V:=100.000, z1, wi_tGripper, \WObj:=handpos;
MoveL t122, v100\V:=100.000, z1, wi_tGripper, \WObj:=handpos;
MoveL t123, v100\V:=100.000, z1, wi_tGripper, \WObj:=handpos;
MoveL t124, v100\V:=100.000, z1, wi_tGripper, \WObj:=handpos;
MoveL t125, v100\V:=100.000, z1, wi_tGripper, \WObj:=handpos;
MoveL t126, v100\V:=100.000, z1, wi_tGripper, \WObj:=handpos;
MoveL t127, v100\V:=100.000, z1, wi_tGripper, \WObj:=handpos;
MoveL t128, v100\V:=100.000, z1, wi_tGripper, \WObj:=handpos;
MoveL t129, v100\V:=100.000, z1, wi_tGripper, \WObj:=handpos;
MoveL t130, v100\V:=100.000, z1, wi_tGripper, \WObj:=handpos;
MoveL t131, v100\V:=100.000, z1, wi_tGripper, \WObj:=handpos;
MoveL t132, v100\V:=100.000, z1, wi_tGripper, \WObj:=handpos;
MoveL t133, v100\V:=100.000, z1, wi_tGripper, \WObj:=handpos;
MoveL t134, v100\V:=100.000, z1, wi_tGripper, \WObj:=handpos;
MoveL t135, v100\V:=100.000, z1, wi_tGripper, \WObj:=handpos;
MoveL t136, v100\V:=100.000, z1, wi_tGripper, \WObj:=handpos;
MoveL t137, v100\V:=100.000, z1, wi_tGripper, \WObj:=handpos;
MoveL t138, v100\V:=100.000, z1, wi_tGripper, \WObj:=handpos;
MoveL t139, v100\V:=100.000, z1, wi_tGripper, \WObj:=handpos;
MoveL t140, v100\V:=100.000, z1, wi_tGripper, \WObj:=handpos;
MoveL t141, v100\V:=100.000, z1, wi_tGripper, \WObj:=handpos;
MoveL t142, v100\V:=100.000, z1, wi_tGripper, \WObj:=handpos;
MoveL t143, v100\V:=100.000, z1, wi_tGripper, \WObj:=handpos;
MoveL t144, v100\V:=100.000, z1, wi_tGripper, \WObj:=handpos;
MoveL t145, v100\V:=100.000, z1, wi_tGripper, \WObj:=handpos;
MoveL t146, v100\V:=100.000, z1, wi_tGripper, \WObj:=handpos;
MoveL t147, v100\V:=100.000, z1, wi_tGripper, \WObj:=handpos;
MoveL t148, v100\V:=100.000, z1, wi_tGripper, \WObj:=handpos;
MoveL t149, v100\V:=100.000, z1, wi_tGripper, \WObj:=handpos;
MoveL t150, v100\V:=100.000, z1, wi_tGripper, \WObj:=handpos;
MoveL t151, v100\V:=100.000, z1, wi_tGripper, \WObj:=handpos;
MoveL t152, v100\V:=100.000, z1, wi_tGripper, \WObj:=handpos;
MoveL t153, v100\V:=100.000, z1, wi_tGripper, \WObj:=handpos;
MoveL t154, v100\V:=100.000, z1, wi_tGripper, \WObj:=handpos;
MoveL t155, v100\V:=100.000, z1, wi_tGripper, \WObj:=handpos;
MoveL t156, v100\V:=100.000, z1, wi_tGripper, \WObj:=handpos;
MoveL t157, v100\V:=100.000, z1, wi_tGripper, \WObj:=handpos;
MoveL t158, v100\V:=100.000, z1, wi_tGripper, \WObj:=handpos;
MoveL t159, v100\V:=100.000, z1, wi_tGripper, \WObj:=handpos;
MoveL t160, v100\V:=100.000, z1, wi_tGripper, \WObj:=handpos;
MoveL t161, v100\V:=100.000, z1, wi_tGripper, \WObj:=handpos;
MoveL t162, v100\V:=100.000, z1, wi_tGripper, \WObj:=handpos;
MoveL t163, v100\V:=100.000, z1, wi_tGripper, \WObj:=handpos;
MoveL t164, v100\V:=100.000, z1, wi_tGripper, \WObj:=handpos;
MoveL t165, v100\V:=100.000, z1, wi_tGripper, \WObj:=handpos;
MoveL t166, v100\V:=100.000, z1, wi_tGripper, \WObj:=handpos;
MoveL t167, v100\V:=100.000, z1, wi_tGripper, \WObj:=handpos;
MoveL t168, v100\V:=100.000, z1, wi_tGripper, \WObj:=handpos;
MoveL t169, v100\V:=100.000, z1, wi_tGripper, \WObj:=handpos;
MoveL t170, v100\V:=100.000, z1, wi_tGripper, \WObj:=handpos;
MoveL t171, v100\V:=100.000, z1, wi_tGripper, \WObj:=handpos;
MoveL t172, v100\V:=100.000, z1, wi_tGripper, \WObj:=handpos;
MoveL t173, v100\V:=100.000, z1, wi_tGripper, \WObj:=handpos;
MoveL t174, v100\V:=100.000, z1, wi_tGripper, \WObj:=handpos;
MoveL t175, v100\V:=100.000, z1, wi_tGripper, \WObj:=handpos;
MoveL t176, v100\V:=100.000, z1, wi_tGripper, \WObj:=handpos;
MoveL t177, v100\V:=100.000, z1, wi_tGripper, \WObj:=handpos;
MoveL t178, v100\V:=100.000, z1, wi_tGripper, \WObj:=handpos;
MoveL t179, v100\V:=100.000, z1, wi_tGripper, \WObj:=handpos;
MoveL t180, v100\V:=100.000, z1, wi_tGripper, \WObj:=handpos;
MoveL t181, v100\V:=100.000, z1, wi_tGripper, \WObj:=handpos;
MoveL t182, v100\V:=100.000, z1, wi_tGripper, \WObj:=handpos;
MoveL t183, v100\V:=100.000, z1, wi_tGripper, \WObj:=handpos;
MoveL t184, v100\V:=100.000, z1, wi_tGripper, \WObj:=handpos;
MoveL t185, v100\V:=100.000, z1, wi_tGripper, \WObj:=handpos;
MoveL t186, v100\V:=100.000, z1, wi_tGripper, \WObj:=handpos;
MoveL t187, v100\V:=100.000, z1, wi_tGripper, \WObj:=handpos;
MoveL t188, v100\V:=100.000, z1, wi_tGripper, \WObj:=handpos;
MoveL t189, v100\V:=100.000, z1, wi_tGripper, \WObj:=handpos;
MoveL t190, v100\V:=100.000, z1, wi_tGripper, \WObj:=handpos;
MoveL t191, v100\V:=100.000, z1, wi_tGripper, \WObj:=handpos;
MoveL t192, v100\V:=100.000, z1, wi_tGripper, \WObj:=handpos;
MoveL t193, v100\V:=100.000, z1, wi_tGripper, \WObj:=handpos;
MoveL t194, v100\V:=100.000, z1, wi_tGripper, \WObj:=handpos;
MoveL t195, v100\V:=100.000, z1, wi_tGripper, \WObj:=handpos;
MoveL t196, v100\V:=100.000, z1, wi_tGripper, \WObj:=handpos;
MoveL t197, v100\V:=100.000, z1, wi_tGripper, \WObj:=handpos;
MoveL t198, v100\V:=100.000, z1, wi_tGripper, \WObj:=handpos;
MoveL t199, v100\V:=100.000, z1, wi_tGripper, \WObj:=handpos;

ENDPROC
ENDMODULE
